// TIA Portal project "Cau2" (V16)

(* hardware
DEVICE "S7-1200 station_1"  S7-1200 Station
   slot 0: "Rack_0"  S7-1200 Rack  Rack  V1.0
   slot 1: "PLC_1"  CPU 1212C DC/DC/DC  6ES7 212-1AE40-0XB0  V4.3
   slot 2: "DI 16/DQ 16x24VDC_1"  6ES7 223-1BL32-0XB0  V2.0
   slot 3: "DQ 16xRelay_1"  SM 1222 DQ16 x relay  6ES7 222-1HH32-0XB0  V2.0
*)

// ===== PLC "PLC_1"  CPU 1212C DC/DC/DC =====

VAR_GLOBAL   // PLC tag table "Default tag table"
   "Start" AT %I8.3 : Bool;
   "Stop" AT %I8.2 : Bool;
   "Biến giữ chương trình" AT %M0.0 : Bool;
   "KM1" AT %Q0.0 : Bool;
   "KM2" AT %Q0.1 : Bool;
   "KM3" AT %Q0.2 : Bool;
   "KM4" AT %Q0.3 : Bool;
END_VAR

// folder: System blocks/Program resources

DATA_BLOCK "T1"   // DB1
{ S7_Optimized_Access := 'TRUE' }
AUTHOR : Simatic
FAMILY : IEC
NAME : IEC_TMR
VERSION : 1.0
// stored: InstanceOfName IEC_TIMER
"IEC_TIMER"
BEGIN
END_DATA_BLOCK

DATA_BLOCK "T2"   // DB2
{ S7_Optimized_Access := 'TRUE' }
AUTHOR : Simatic
FAMILY : IEC
NAME : IEC_TMR
VERSION : 1.0
// stored: InstanceOfName IEC_TIMER
"IEC_TIMER"
BEGIN
END_DATA_BLOCK

DATA_BLOCK "T3"   // DB3
{ S7_Optimized_Access := 'TRUE' }
AUTHOR : Simatic
FAMILY : IEC
NAME : IEC_TMR
VERSION : 1.0
// stored: InstanceOfName IEC_TIMER
"IEC_TIMER"
BEGIN
END_DATA_BLOCK

// folder: (top level)

ORGANIZATION_BLOCK "Main"   // OB1, LAD, ProgramCycle
TITLE = "Main Program Sweep (Cycle)"
{ S7_Optimized_Access := 'TRUE' }
VERSION : 0.1
   VAR_INPUT
      Initial_Call : Bool;   // Initial call of this OB
      Remanence : Bool;   // =True, if remanent data are available
   END_VAR
BEGIN

REGION Network 1
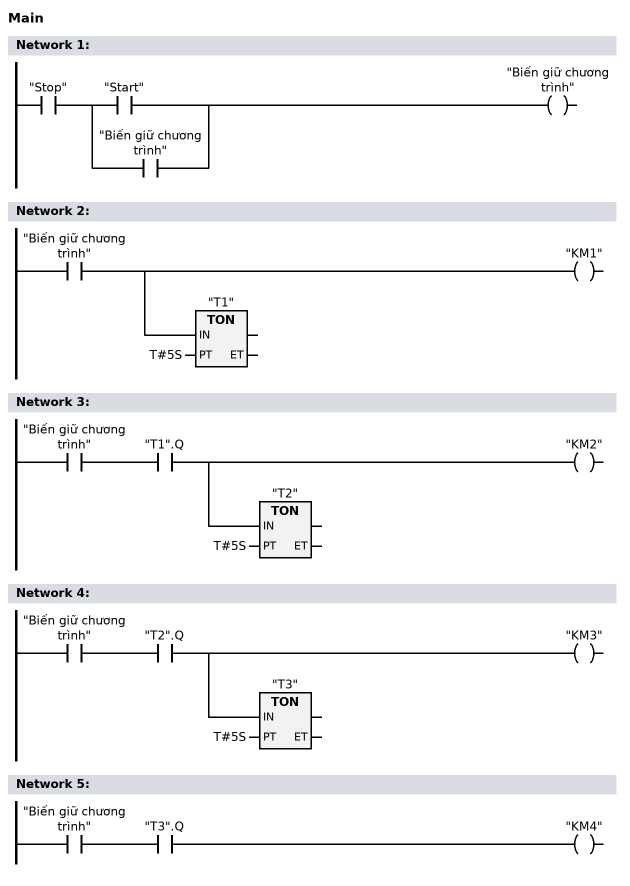
   RUNG wire#powerrail
      Contact( "Stop" )
      wire#w1
      Contact( "Start" )
      wire#w2
      Coil( "Biến giữ chương trình" )
   END_RUNG
   RUNG wire#w1
      Contact( "Biến giữ chương trình" )
   END_RUNG wire#w2
   // the same network as SCL:
   "Biến giữ chương trình" := "Stop" AND ("Start" OR "Biến giữ chương trình");
END_REGION

REGION Network 2
   "KM1" := "Biến giữ chương trình";
   "T1".TON(IN := "Biến giữ chương trình", PT := T#5S);
END_REGION

REGION Network 3
   "KM2" := "Biến giữ chương trình" AND "T1".Q;
   "T2".TON(IN := "KM2", PT := T#5S);
END_REGION

REGION Network 4
   "KM3" := "Biến giữ chương trình" AND "T2".Q;
   "T3".TON(IN := "KM3", PT := T#5S);
END_REGION

REGION Network 5
   RUNG wire#powerrail
      Contact( "Biến giữ chương trình" )
      Contact( "T3".Q )
      Coil( "KM4" )
   END_RUNG
   // the same network as SCL:
   "KM4" := "Biến giữ chương trình" AND "T3".Q;
END_REGION
END_ORGANIZATION_BLOCK